# EPICS autosave request: support/pilatus/1-6/pilatusApp/Db/pilatus_settings.req
$(DET)IMGPATH-SET
$(DET)FILENAME
$(DET)EXPTIME-SET
$(DET)NIMAGE-SET
$(DET)NEXPFRM-SET
$(DET)DELAY-SET
$(DET)TRIMFILE
